Universal Robots PolyScope program: MT_SFF_Simulation.urp

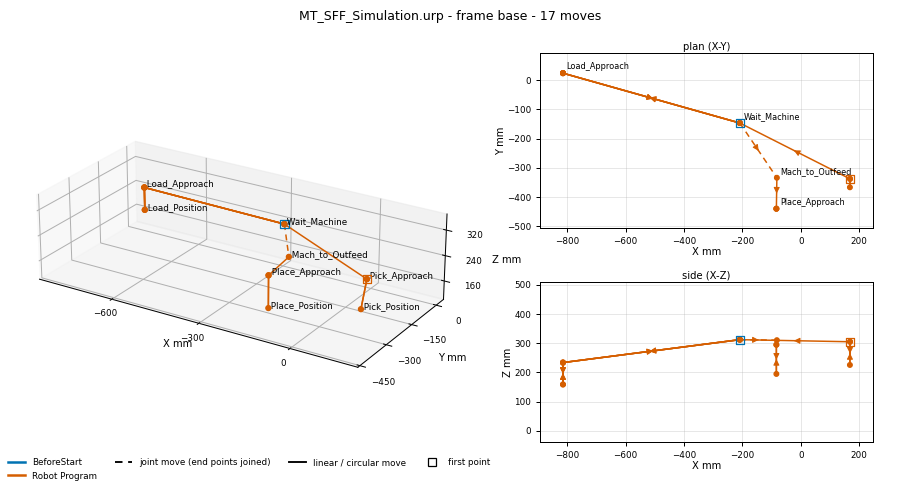
[picture p0: tool path of MT_SFF_Simulation.urp in frame base, 17 of 17 moves have a stored position in this frame; points joined in program order, loops and branches not executed]
Program MT_SFF_Simulation (createdIn=3.5.1.10661 lastSavedIn=5.1.0.40195 robotSerialNumber=2014359999 directory=/home/ur/ursim-current/programs/Machine Tending/FullSimulationDownload/SFF installation=default)
Calibrated DH parameters: a=[0, -0.425, -0.3922, 0, 0, 0]; d=[0.1625, 0, 0, 0.1333, 0.0997, 0.0996]; alpha=[1.570796, 0, 0, 1.570796, -1.570796, 0]; deltaTheta=[0, 0, 0, 0, 0, 0]
BeforeStart
  MoveJ speed 60 deg/s, acceleration 80 deg/s^2 (useActiveTCP=false) feature=Base
    Waypoint Wait_Machine: TCP in base x=-208.762 y=-146.481 z=312.267 mm, rx=2.9475 ry=1.087 rz=0 rad; joints [-15.789, -147.455, 140.244, -111.828, -53.977, 43.352] deg; TCP offset x=70 y=0 z=80 mm, rx=0 ry=0.7854 rz=0 rad
  Folder Status
    Infeed_Ready := True   [initializeExpression=False]
    Outfeed_Ready := True   [initializeExpression=False]
  Folder Initialization
    Call Tool_1_Off
Robot Program (runOnlyOnce=false)
  Wait Condition expression=Infeed_Ready≟ True
  Folder INFEED - Fixed
    MoveL speed 1000 mm/s, acceleration 2500 mm/s^2 (useActiveTCP=false) tcp=TCP; feature=Base
      Waypoint Pick_Approach: TCP in base x=168.331 y=-337.561 z=305.093 mm, rx=2.0348 ry=2.0328 rz=-0.3642 rad; joints [97.405, -116.228, 128.726, -122.307, -92.836, 96.964] deg; TCP offset x=0 y=0 z=100 mm, rx=0 ry=0 rz=0 rad
      Waypoint Pick_Position: TCP in base x=167.871 y=-366.461 z=225.69 mm, rx=2.0348 ry=2.0328 rz=-0.3642 rad; joints [96.648, -106.517, 135.586, -138.911, -92.579, 96.252] deg
      Call Tool_1_On
      Waypoint Pick_Approach: TCP in base x=168.331 y=-337.561 z=305.093 mm, rx=2.0348 ry=2.0328 rz=-0.3642 rad; joints [97.405, -116.228, 128.726, -122.307, -92.836, 96.964] deg
      Waypoint Wait_Machine: TCP in base x=-208.762 y=-146.481 z=312.267 mm, rx=2.9475 ry=1.087 rz=0 rad; joints [-15.789, -147.455, 140.244, -111.828, -53.977, 43.352] deg; TCP offset x=70 y=0 z=80 mm, rx=0 ry=0.7854 rz=0 rad
  Folder MACHINE
    Wait DigitalInput pin=GP_bool_in[1]; digitalValue=1
    Folder LOAD
      MoveL speed 1000 mm/s, acceleration 2500 mm/s^2 (useActiveTCP=false) tcp=TCP; feature=Base
        Waypoint Load_Approach: motionParameters(blendRadius=0.05); TCP in base x=-814.054 y=24.13 z=233.886 mm, rx=3.1416 ry=0 rz=0 rad; joints [-12.297, -47.749, 68.099, -154.684, -81.338, 81.237] deg; TCP offset x=70 y=0 z=80 mm, rx=0 ry=0.7854 rz=0 rad
        Waypoint Load_Position: TCP in base x=-814.054 y=24.13 z=158.886 mm, rx=3.1416 ry=0 rz=0 rad; joints [-11.118, -41.062, 53.307, -102.245, -90, 78.882] deg; TCP offset x=0 y=0 z=100 mm, rx=0 ry=0 rz=0 rad
        Call Holding_On
        Call Tool_1_Off
        Waypoint Load_Approach: TCP in base x=-814.054 y=24.13 z=233.886 mm, rx=3.1416 ry=0 rz=0 rad; joints [-12.297, -47.749, 68.099, -154.684, -81.338, 81.237] deg; TCP offset x=70 y=0 z=80 mm, rx=0 ry=0.7854 rz=0 rad
        Waypoint Wait_Machine: TCP in base x=-208.762 y=-146.481 z=312.267 mm, rx=2.9475 ry=1.087 rz=0 rad; joints [-15.789, -147.455, 140.244, -111.828, -53.977, 43.352] deg; TCP offset x=70 y=0 z=80 mm, rx=0 ry=0.7854 rz=0 rad
      Set DigitalOutput pin=GP_bool_out[1]; digitalValue=1
      Wait DigitalInput pin=GP_bool_in[1]; digitalValue=0
      Set DigitalOutput pin=GP_bool_out[1]; digitalValue=0
    Wait DigitalInput pin=GP_bool_in[0]; digitalValue=1
    Folder UNLOAD
      MoveL speed 1000 mm/s, acceleration 2500 mm/s^2 (useActiveTCP=false) tcp=TCP; feature=Base
        Waypoint Load_Approach: motionParameters(blendRadius=0.05); TCP in base x=-814.054 y=24.13 z=233.886 mm, rx=3.1416 ry=0 rz=0 rad; joints [-12.297, -47.749, 68.099, -154.684, -81.338, 81.237] deg; TCP offset x=70 y=0 z=80 mm, rx=0 ry=0.7854 rz=0 rad
        Waypoint Load_Position: TCP in base x=-814.054 y=24.13 z=158.886 mm, rx=3.1416 ry=0 rz=0 rad; joints [-11.118, -41.062, 53.307, -102.245, -90, 78.882] deg; TCP offset x=0 y=0 z=100 mm, rx=0 ry=0 rz=0 rad
        Call Tool_1_On
        Call Holding_Off
        Waypoint Load_Approach: TCP in base x=-814.054 y=24.13 z=233.886 mm, rx=3.1416 ry=0 rz=0 rad; joints [-12.297, -47.749, 68.099, -154.684, -81.338, 81.237] deg; TCP offset x=70 y=0 z=80 mm, rx=0 ry=0.7854 rz=0 rad
        Waypoint Wait_Machine: TCP in base x=-208.762 y=-146.481 z=312.267 mm, rx=2.9475 ry=1.087 rz=0 rad; joints [-15.789, -147.455, 140.244, -111.828, -53.977, 43.352] deg; TCP offset x=70 y=0 z=80 mm, rx=0 ry=0.7854 rz=0 rad
      Set DigitalOutput pin=GP_bool_out[0]; digitalValue=1
      Wait DigitalInput pin=GP_bool_in[0]; digitalValue=0
      Set DigitalOutput pin=GP_bool_out[0]; digitalValue=0
  Wait Condition expression=Outfeed_Ready≟ True
  Folder OUTFEED - Fixed
    MoveJ speed 120 deg/s, acceleration 150 deg/s^2 (useActiveTCP=false) tcp=TCP; feature=Base
      Waypoint Mach_to_Outfeed: motionParameters(blendRadius=0.05); TCP in base x=-82.05 y=-333.74 z=310.5 mm, rx=2.2183 ry=2.2183 rz=-0.0069 rad; joints [53.231, -114.218, 120.145, -96.213, -89.785, 53.233] deg; TCP offset x=0 y=0 z=100 mm, rx=0 ry=0 rz=0 rad
    MoveL speed 250 mm/s, acceleration 1200 mm/s^2 (useActiveTCP=false) tcp=TCP; feature=Base
      Waypoint Place_Approach: TCP in base x=-83.738 y=-439.7 z=294.892 mm, rx=-2.2214 ry=-2.2214 rz=0 rad; joints [61.891, -97.334, 110.53, -103.196, -90, 61.891] deg
      Waypoint Place_Position: TCP in base x=-83.739 y=-439.699 z=194.954 mm, rx=-2.2214 ry=-2.2214 rz=0 rad; joints [61.891, -91.887, 121.318, -119.431, -90, 61.891] deg
      Call Tool_1_Off
      Waypoint Place_Approach: TCP in base x=-83.738 y=-439.7 z=294.892 mm, rx=-2.2214 ry=-2.2214 rz=0 rad; joints [61.891, -97.334, 110.53, -103.196, -90, 61.891] deg
SubProgram  [hidden by the author, left out]
SubProgram  [hidden by the author, left out]
SubProgram  [hidden by the author, left out]
SubProgram  [hidden by the author, left out]
SubProgram Tool_1_Off [hidden by the author, left out]
SubProgram Tool_1_On [hidden by the author, left out]
SubProgram Holding_On [hidden by the author, left out]
SubProgram Holding_Off [hidden by the author, left out]
